FUNCTION_BLOCK AxesPower IMPLEMENTS ITask
VAR_INPUT
END_VAR
VAR_OUTPUT
END_VAR
VAR
	_busy : BOOL;
	_error : BOOL;
	_done : BOOL;
	State : INT;
	_axis : REFERENCE TO Tc2_MC2.AXIS_REF;
END_VAR

CASE State OF
	0:
	1:
END_CASE

{warning 'add method implementation '}
METHOD Abort : BOOL
END_METHOD

{warning 'add property implementation'}
PROPERTY Busy : BOOL
GET
Busy := _busy;
END_GET
END_PROPERTY

{warning 'add property implementation'}
PROPERTY Done : BOOL
GET
Done := _done;
END_GET
END_PROPERTY

{warning 'add property implementation'}
PROPERTY Error : BOOL
GET
Error := _error;
END_GET
END_PROPERTY

METHOD FB_init : BOOL
VAR_INPUT
	bInitRetains : BOOL; // if TRUE, the retain variables are initialized (warm start / cold start)
	bInCopyCode : BOOL;  // if TRUE, the instance afterwards gets moved into the copy code (online change)
	axis : reference TO AXIS_REF;
END_VAR
_axis REF= axis;
END_METHOD

END_FUNCTION_BLOCK

(* stored: Version 1.1.0.1, ProductVersion 3.1.4024.6
   POU AxesPower: Id {23d1f2a2-599f-44a8-80a3-c75c682185de}, SpecialFunc None
   Method Abort: Id {e1aa31b7-91fd-4a85-bda7-7ec456f14df3}
   Property Busy: Id {279189bd-55f4-4622-ad19-ce4053f31ada}
   Get Get: Id {09f5299d-99cd-486a-bfa5-b42ba97b116d}
   Property Done: Id {33e9adaa-f326-44e7-b147-e42057d89ae1}
   Get Get: Id {9b0dd4aa-7eb9-48f1-8128-1a9373e8c013}
   Property Error: Id {4490fc92-1c23-4dbb-955e-41cc66763287}
   Get Get: Id {43f61c88-8fc7-47e6-bf43-eaa98b4f4aa1}
   Method FB_init: Id {df919bb3-3c47-47f1-a703-c7dae88ab8fa} *)
